(* PLC project Tc2_Utilities.FB_RegSetValue Demo, tc3-libraries-kb TwinCAT 3.1 *)
(* stored: creationDateTime 2026-05-11T00:00:00, modificationDateTime 2026-05-11T00:00:00 *)

PROGRAM P_Demo_FB_RegSetValue
  VAR
    fbFB_RegSetValue : FB_RegSetValue;  (* FB_RegSetValue 实例 *)
    sNetId : T_AmsNetId;
    sSubKey : T_MaxString;
    sValName : T_MaxString;
    eValType : E_RegValueType;
    cbData : UDINT;
    pData : POINTER TO BYTE;
    bExecute : BOOL;
    tTimeOut : TIME := DEFAULT_ADS_TIMEOUT;
    bBusy : BOOL;
    bError : BOOL;
    nErrId : UDINT;
    cbWrite : UDINT;
  END_VAR

// =============================================================================
// 场景：commissioning 配置注册表。
// 价值：脚本化。
// 验证：写一个测试键，用 FB_RegQueryValue 读回应一致。
// 验证步骤：
//   1. 右键 PLC 项目 → Import PLCopenXML → 选本文件
//   2. 引用 Tc2_Utilities（References → Add library）
//   3. 编译 → 登录 → 运行；按上方『验证』行的指示在线写值观察
// =============================================================================

// 单次完整调用形式（所有 VAR_INPUT 显式赋值）
fbFB_RegSetValue(
    sNetId := sNetId,
    sSubKey := sSubKey,
    sValName := sValName,
    eValType := eValType,
    cbData := cbData,
    pData := pData,
    bExecute := bExecute,
    tTimeOut := tTimeOut,
    bBusy => bBusy,
    bError => bError,
    nErrId => nErrId,
    cbWrite => cbWrite
);
END_PROGRAM
